TYPE ST_Auto_Status :
STRUCT
END_STRUCT
END_TYPE

(* stored: Version 1.1.0.1, ProductVersion 3.1.4024.13
   DUT ST_Auto_Status: Id {71a8bc26-8c44-42c1-9bb5-05e42c3b29ae} *)
